{attribute 'GeneratedUsingTerminal: AT2041-0250-0018'}
{attribute addProperty BoxType "AT2041-0250-0018"}
{attribute addProperty Id "A_0104_AT2042_5250_0019_AT2042_5250AT2042_01D6DEDF80"}
{attribute addProperty CRC "3254445086"}
{attribute addProperty Size "80"}
TYPE A_0040_AT2041_0250_0018_C1FAE41E EXTENDS AT2041_86175B41 :
STRUCT
	{attribute addProperty Name "A_0104_AT2042_5250_0019_AT2042_5250"}
	A_0104_AT2042_5250_0019_AT2042_5250 : AT2042_01D6DEDF;
END_STRUCT
END_TYPE

(* stored: Version 1.2.0.0, ProductVersion 3.1.4024.9
   DUT A_0040_AT2041_0250_0018_C1FAE41E: Id {29c701d6-e160-43a4-8833-c05887e14e78} *)
